FUNCTION_BLOCK FB_TiltControlEmulation 
VAR_INPUT	
	Config					: ST_CFG_TiltPositionEmu; // emulation config	
	DriveRun_Up				: BOOL;
	DriveRun_Down      		: BOOL;
END_VAR

VAR_OUTPUT
	Lift_Pos_Up				: BOOL;
	Lift_Pos_Down			: BOOL;
	Lift_Pos_Middle			: BOOL;
	
END_VAR

VAR
	ActualPosition			: INT :=0;
END_VAR

// When lift is moving
IF DriveRun_Up THEN
	IF ActualPosition < Config.Position_Max_Up THEN
	ActualPosition := ActualPosition + 1;
	END_IF
END_IF

IF DriveRun_Down THEN
	IF ActualPosition > Config.Position_Max_Down THEN
	ActualPosition := ActualPosition - 1;
	END_IF
END_IF


// Update positions
IF ActualPosition = Config.Position_Down THEN
	 Lift_Pos_Down := TRUE;
ELSIF ActualPosition = Config.Position_Up THEN
	 Lift_Pos_Up := TRUE;
ELSIF ActualPosition = Config.Position_Middle THEN
	Lift_Pos_Middle := TRUE;
ELSE  	
	Lift_Pos_Down := FALSE;
	Lift_Pos_Up := FALSE;
	Lift_Pos_Middle := FALSE;
END_IF

END_FUNCTION_BLOCK

(* stored: Version 1.1.0.1, ProductVersion 3.1.4024.9
   POU FB_TiltControlEmulation: Id {6a616511-852d-4cac-ba9c-7a01278c94cc}, SpecialFunc None *)
